(* PLC project Unnamed, Unknown Unnamed 1 *)
(* stored: creationDateTime 2019-08-06T14:23:42, modificationDateTime 2021-01-19T09:52:38 *)

PROGRAM MainStuff
  VAR
    TargetPressure : HMI_INT;
    selection : HMI_INT;
  END_VAR

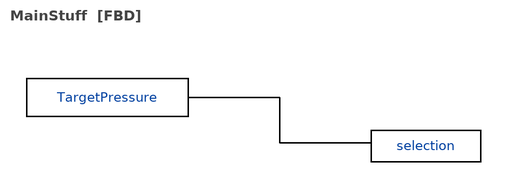
(* FBD diagram, written out as Structured Text *)
selection := TargetPressure;
END_PROGRAM

CONFIGURATION config
  RESOURCE resource1 ON PLC
    TASK task0(INTERVAL := T#20ms, PRIORITY := 0);
    PROGRAM instance0 WITH task0 : MainStuff;
  END_RESOURCE
END_CONFIGURATION
